{attribute 'GeneratedUsingTerminal: EK1960-0000-0019'}
{attribute addProperty BoxType "EK1960-0000-0019"}
{attribute addProperty Id "OutputsOutputs_63C46CC828"}
{attribute addProperty CRC "3897236224"}
{attribute addProperty Size "28"}
TYPE Module_2_FSOUT_E84B1B00 :
STRUCT
	{attribute addProperty Name "Outputs"}
	Outputs  : Outputs_63C46CC8;
END_STRUCT
END_TYPE

(* stored: Version 1.2.0.0, ProductVersion 3.1.4024.9
   DUT Module_2_FSOUT_E84B1B00: Id {50c7dd67-c63a-448e-8b54-0820d98bac80} *)
